(* IEC 61131-3 sources: repolevel_ST_code_completion/dataset/project_code/轴控/FB105_轴控制集/FB50_虚轴控制/FB102_隐含检查, 10 files *)

(* ---- CheckBounds.st ---- *)
// 隐式生成代码:不需要编辑
FUNCTION CheckBounds : DINT
VAR_INPUT
	index, lower, upper: DINT;
END_VAR

// 隐式生成代码:只是实现代码的建议
IF  index < lower THEN
	CheckBounds := lower;
ELSIF  index > upper THEN
	CheckBounds := upper;
ELSE
	CheckBounds := index;
END_IF

(*还可以设置断点,日志信息或其他.比如在异常处停止:
Add CmpApp.library, SysExcept.library and SysTypes2_Itf as newest.
Declaration:
VAR
    _pApp : POINTER TO CmpApp.APPLICATION;
    _result   : SysTypes.RTS_IEC_RESULT;
END_VAR

Implementation:
_pApp := AppGetCurrent(pResult:=_result);
IF  index < lower THEN
        CheckBounds := lower;
        IF _pApp <> 0 THEN
                AppGenerateException(pApp:=_pApp, ulException:=RtsExceptions.RTSEXCPT_ARRAYBOUNDS);
        END_IF
ELSIF  index > upper THEN
        CheckBounds := upper;
        IF _pApp <> 0 THEN
                AppGenerateException(pApp:=_pApp,   ulException:=RtsExceptions.RTSEXCPT_ARRAYBOUNDS);
        END_IF
ELSE
        CheckBounds := index;
END_IF
*)

(* ---- CheckDivDInt.st ---- *)
// 隐式生成代码:不需要编辑
FUNCTION CheckDivDInt : DINT
VAR_INPUT
	divisor:DINT;
END_VAR

// 隐式生成代码:只是实现代码的建议
IF divisor = 0 THEN
	CheckDivDInt:=1;
ELSE
	CheckDivDInt:=divisor;
END_IF;

(* ---- CheckDivLInt.st ---- *)
// 隐式生成代码:不需要编辑
FUNCTION CheckDivLInt : LINT
VAR_INPUT
	divisor:LINT;
END_VAR

// 隐式生成代码:只是实现代码的建议
IF divisor = 0 THEN
	CheckDivLInt:=1;
ELSE
	CheckDivLInt:=divisor;
END_IF;

(* ---- CheckDivLReal.st ---- *)
// 隐式生成代码:不需要编辑
FUNCTION CheckDivLReal : LREAL
VAR_INPUT
	divisor:LREAL;
END_VAR

// 隐式生成代码:只是实现代码的建议
IF divisor = 0 THEN
	CheckDivLReal:=1;
ELSE
	CheckDivLReal:=divisor;
END_IF;

(* ---- CheckDivReal.st ---- *)
// 隐式生成代码:不需要编辑
FUNCTION CheckDivReal : REAL
VAR_INPUT
	divisor:REAL;
END_VAR

// 隐式生成代码:只是实现代码的建议
IF divisor = 0 THEN
	CheckDivReal:=1;
ELSE
	CheckDivReal:=divisor;
END_IF;

(* ---- CheckLRangeSigned.st ---- *)
// 隐式生成代码:不需要编辑
FUNCTION CheckLRangeSigned : LINT
VAR_INPUT
	value, lower, upper: LINT;
END_VAR

// 隐式生成代码:只是实现代码的建议
IF (value < lower) THEN
	CheckLRangeSigned := lower;
ELSIF(value > upper) THEN
	CheckLRangeSigned := upper;
ELSE
	CheckLRangeSigned := value;
END_IF

(* ---- CheckLRangeUnsigned.st ---- *)
// 隐式生成代码:不需要编辑
FUNCTION CheckLRangeUnsigned : ULINT
VAR_INPUT
	value, lower, upper: ULINT;
END_VAR

// 隐式生成代码:只是实现代码的建议
IF (value < lower) THEN
	CheckLRangeUnsigned := lower;
ELSIF(value > upper) THEN
	CheckLRangeUnsigned := upper;
ELSE
	CheckLRangeUnsigned := value;
END_IF

(* ---- CheckPointer.st ---- *)
// 隐式生成代码:不需要编辑
FUNCTION CheckPointer : POINTER TO BYTE
VAR_INPUT
	ptToTest : POINTER TO BYTE; // 指针的目标地址
	iSize : DINT;		         //指针指向的类型大小.(例如:POINTER TO ARRAY [0..9] OF INT为20)
	iGran : DINT;		        // 指针访问的粒度,即指针指向的类型中最大的非结构数据类型的大小.(例如: POINTER TO ARRAY [0..9] OF INT为2)
	bWrite: BOOL;		        // 标识读或写权限.TRUE = 写权限.
END_VAR

// 没有标准的实现方式.在此处输入代码
CheckPointer := ptToTest;

(* ---- CheckRangeSigned.st ---- *)
// 隐式生成代码:不需要编辑
FUNCTION CheckRangeSigned : DINT
VAR_INPUT
	value, lower, upper: DINT;
END_VAR

// 隐式生成代码:只是实现代码的建议
IF (value < lower) THEN
	CheckRangeSigned := lower;
ELSIF(value > upper) THEN
	CheckRangeSigned := upper;
ELSE
	CheckRangeSigned := value;
END_IF

(* ---- CheckRangeUnsigned.st ---- *)
// 隐式生成代码:不需要编辑
FUNCTION CheckRangeUnsigned : UDINT
VAR_INPUT
	value, lower, upper: UDINT;
END_VAR

// 隐式生成代码:只是实现代码的建议
IF (value < lower) THEN
	CheckRangeUnsigned := lower;
ELSIF(value > upper) THEN
	CheckRangeUnsigned := upper;
ELSE
	CheckRangeUnsigned := value;
END_IF
